Yaskawa INFORM job: 20231012JOHN.JBI

/JOB
//NAME 20231012JOHN
//POS
///NPOS 6,0,0,0,0,0
///TOOL 5
///POSTYPE PULSE
///PULSE
C00000=-1,-50477,-58433,3,-74929,486
C00001=-26297,12121,-59031,-60331,-33729,36347
C00002=-28379,15703,-65247,-78012,-32860,47340
C00003=-16153,12304,-69817,-85250,-28416,47472
C00004=-16152,9575,-68570,-80080,-28658,44699
C00005=-2,-50477,-58433,4,-74930,485
//INST
///DATE 2024/03/04 14:57
///ATTR SC,RW
///GROUP1 RB1
NOP
MOVJ C00000 VJ=10.00
MOVJ C00001 VJ=8.00
MOVJ C00002 VJ=2.00
ARCON AC=80 AVP=100
DOUT OT#(17) ON
TIMER T=2.00
MOVL C00003 V=2.0
DOUT OT#(17) OFF
ARCOF
MOVJ C00004 VJ=2.00
MOVJ C00005 VJ=8.00
END
